// TIA Portal V16 export
// export: Created 2023-03-29T11:04:28.7082875Z, ExportSetting WithDefaults, DisplayName Totally Integrated Automation Portal, DisplayVersion V16 Update 6, DisplayName TIA Portal Version Control Interface, DisplayVersion V16 Update 2, DisplayName TIA Portal Openness, DisplayVersion V16 Update 6, DisplayName STEP 7 Professional, DisplayVersion V16 Update 6, DisplayName STEP 7 Safety, DisplayVersion V16, DisplayName WinCC Advanced, DisplayVersion V16 Update 6
FUNCTION_BLOCK "WatchDog HMI"   // FB12, LAD
TITLE = WatchDog HMI
{ S7_Optimized_Access := 'TRUE' }
AUTHOR : rtecmer
VERSION : 0.1
// Kontrola komunikacji PLC z HMI.  Wartość w zmiennej w instancji "Dane_ComunicationControlHMI".tempCoordinationHMIRS5 jest inkrementowana przez PLC i co minutę skrypt z HMI wartość zeruje. Jeśli błąd kumunikacj to wartość jest inkrementowana do max zmiennej. Przy wartości 70 ustawiany jest bit alarmu dla PLC, że btrak komunikacji z HMI
// HMI na podstawie błędu systemowego 190011 komonikuje w tabeli alarmów o braku komunikacji
// stored: AutoNumber true, IsIECCheckEnabled false, IsRetainMemResEnabled false, MemoryReserve 500, SetENOAutomatically false, UDAEnableTagReadback false
   VAR_TEMP   // added for the SCL form of the ladder/FBD networks
      _w1 : Bool;
      _w2 : Bool;
   END_VAR
BEGIN

REGION Network 1: WatchDog HMI
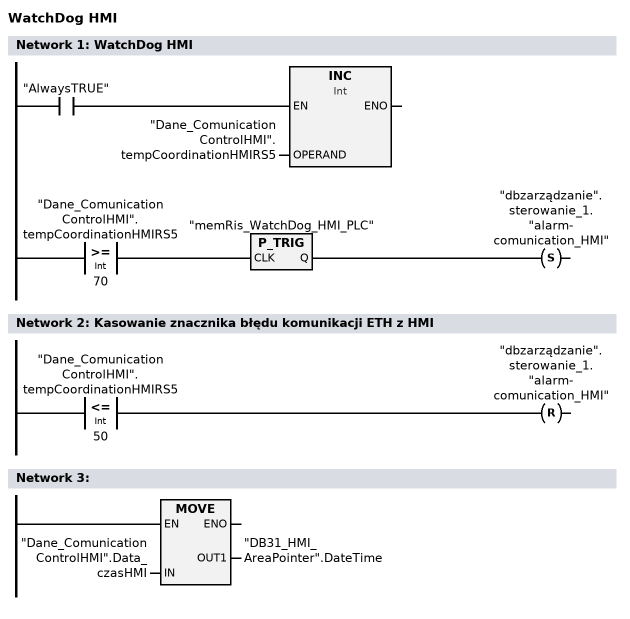
   RUNG wire#powerrail
      Contact( "AlwaysTRUE" )
      { S7_Templates := "DestType := Int" } Inc( "Dane_ComunicationControlHMI".tempCoordinationHMIRS5 )
   END_RUNG
   RUNG wire#powerrail
      { S7_Templates := "SrcType := Int" } GE_Contact(in1 := "Dane_ComunicationControlHMI".tempCoordinationHMIRS5, in2 := 70)
      P_Trig( "memRis_WatchDog_HMI_PLC" )
      S_Coil( "dbzarządzanie".sterowanie_1."alarm-comunication_HMI" )
   END_RUNG
   // the same network as SCL:
   IF "AlwaysTRUE" THEN
       "Dane_ComunicationControlHMI".tempCoordinationHMIRS5 := "Dane_ComunicationControlHMI".tempCoordinationHMIRS5 + 1;
   END_IF;
   #_w1 := "Dane_ComunicationControlHMI".tempCoordinationHMIRS5 >= 70;
   #_w2 := #_w1 AND NOT "memRis_WatchDog_HMI_PLC";   // rising edge
   "memRis_WatchDog_HMI_PLC" := #_w1;
   IF #_w2 THEN "dbzarządzanie".sterowanie_1."alarm-comunication_HMI" := TRUE; END_IF;
END_REGION

REGION Network 2: Kasowanie znacznika błędu komunikacji ETH z HMI
   RUNG wire#powerrail
      { S7_Templates := "SrcType := Int" } LE_Contact(in1 := "Dane_ComunicationControlHMI".tempCoordinationHMIRS5, in2 := 50)
      R_Coil( "dbzarządzanie".sterowanie_1."alarm-comunication_HMI" )
   END_RUNG
   // the same network as SCL:
   IF "Dane_ComunicationControlHMI".tempCoordinationHMIRS5 <= 50 THEN
       "dbzarządzanie".sterowanie_1."alarm-comunication_HMI" := FALSE;
   END_IF;
END_REGION

REGION Network 3
   RUNG wire#powerrail
      Move(in := "Dane_ComunicationControlHMI".Data_czasHMI, out1 => "DB31_HMI_AreaPointer".DateTime)
   END_RUNG
   // the same network as SCL:
   "DB31_HMI_AreaPointer".DateTime := "Dane_ComunicationControlHMI".Data_czasHMI;
END_REGION
END_FUNCTION_BLOCK
